{attribute addProperty BoxType "EL3483-0000-0016"}
{attribute addProperty Id "L1_StatusAT %I*L1_Status_2BC7A2034050L2_StatusAT %I*L2_Status_2BC7A2034050L3_StatusAT %I*L3_Status_2BC7A2034050Total_StatusAT %I*Total_Status_5266C05996120Total_AdvancedAT %I*Total_Advanced_FCA492E91620WcStateAT %I*WcState_98A4DF7520.250InfoDataAT %I*InfoData_BC63D37F80100"}
{attribute addProperty CRC "2860662756"}
{attribute addProperty SizeInBites "314"}
{attribute addProperty SizeInBytes "39.25"}
TYPE EL3483_4A236564 :
STRUCT
	{attribute addProperty Name "L1_Status"}
	L1_Status : L1_Status_2BC7A203;
	{attribute addProperty Name "L2_Status"}
	L2_Status : L2_Status_2BC7A203;
	{attribute addProperty Name "L3_Status"}
	L3_Status : L3_Status_2BC7A203;
	{attribute addProperty Name "Total_Status"}
	Total_Status : Total_Status_5266C059;
	{attribute addProperty Name "Total_Advanced"}
	Total_Advanced : Total_Advanced_FCA492E9;
	{attribute addProperty Name "WcState"}
	WcState : WcState_98A4DF75;
	{attribute addProperty Name "InfoData"}
	InfoData : InfoData_BC63D37F;
END_STRUCT
END_TYPE

(* stored: Version 1.2.0.0, ProductVersion 3.1.4024.9
   DUT EL3483_4A236564: Id {5dcbdd7f-c1c8-461f-b8ef-badb12898794} *)
